{attribute 'GeneratedUsingTerminal: EK1122-0000-0018'}
{attribute addProperty BoxType "EK1122-0000-0018"}
{attribute addProperty Id "Beckhoff_EL1xxxsub_EK1100EK1100_1FC0878B2"}
{attribute addProperty CRC "1293288365"}
{attribute addProperty Size "2"}
TYPE Beckhoff_EL1xxxEK1122_4D1603AD EXTENDS EK1122_1FC0878B :
STRUCT
	{attribute addProperty Name "Beckhoff EL1xxxsub EK1100"}
	{attribute addProperty PreviousPort "Beckhoff EL1xxxEK1122 : D"}
	Beckhoff_EL1xxxsub_EK1100 : EK1100_1FC0878B;
END_STRUCT
END_TYPE

(* stored: Version 1.2.0.0, ProductVersion 3.1.4024.9
   DUT Beckhoff_EL1xxxEK1122_4D1603AD: Id {f59a8d9b-5b73-476c-bfc4-92e6991cf966} *)
